Yaskawa INFORM job: R1_Y(FRONIUS).JBI

/JOB
//NAME R1_Y(FRONIUS)
///FOLDERNAME INNE
//POS
///NPOS 2,2,0,0,0,0
///TOOL 0
///POSTYPE PULSE
///PULSE
C00000=99921,65108,66162,21645,87086,33144
C00001=-83767,-40832,-28914,-19990,95000,-28688
BC00000=201708,367639,507762
BC00001=201708,42,507762
//INST
///DATE 2023/10/04 15:16
///ATTR SC,RW
///GROUP1 RB1,BS1
NOP
MOVJ C00000 BC00000 VJ=0.78
MOVJ C00001 BC00001 VJ=0.78
END
